// TIA Portal V17 export
// export: Created 2026-05-13T13:53:19.1407963Z, ExportSetting WithDefaults, DisplayName Totally Integrated Automation Portal, DisplayVersion V17 Update 4, DisplayName TIA Portal Openness, DisplayVersion V17 Update 4, DisplayName TIA Portal Version Control Interface, DisplayVersion V17, DisplayName SINAMICS Startdrive Advanced, DisplayVersion V17, DisplayName SINAMICS Startdrive G130, G150, S120, S150, SINAMICS MV, S210, DisplayVersion V17, DisplayName SINAMICS Startdrive G110M, G120, G120C, G120D, G120P, G115D, DisplayVersion V17, DisplayName STEP 7 Professional, DisplayVersion V17 Update 4, DisplayName STEP 7 Safety, DisplayVersion V17, DisplayName WinCC Professional, DisplayVersion V17 Update 4
VBScript "VBFunction_1"  Type=Sub
  '提示：
  ' 1. 使用 <CTRL+SPACE> 或 <CTRL+I> 快捷键打开含所有对象和函数的列表
  ' 2. 使用 HMI Runtime 对象写入代码。
  '  示例：HmiRuntime.Screens("Screen_1")。
  ' 3. 使用 <CTRL+J> 快捷键创建对象引用。
  '从此位置起写入代码：
